Fanuc KAREL source: ko00137.KL

-- PROVISIONAL review KL for V940-1; original PC SHA256 c9733091d5a9caca642406f4a9e78df2e7f2884af441e8ad751a3b0832e9d3ab
-- Incomplete behavior may be omitted. Consult companion uncertainty JSON. Do not deploy.
PROGRAM KO00137
%NOLOCKGROUP
VAR
  R : REAL
  N : INTEGER
-- UNRESOLVED_DECL CFG type=00001c
-- UNRESOLVED_DECL OUT type=000102
BEGIN
  -- V9_ZERO_TABLE_METADATA_HINT layout=0001; no indexed target words; source/name/runtime held
  -- UNRESOLVED_PC offsets 5-12; opcodes 9D,23
  -- UNRESOLVED_PC offsets 17-28; opcodes 2E,23
  -- UNRESOLVED_PC offsets 33-43; opcodes 9D,22,A5
  -- UNRESOLVED_PC offsets 48-107; opcodes 27,22,22,27,21,64,22,22,22,22,76,7E,4A
  -- UNRESOLVED_PC offsets 112-116; opcodes 7F
END KO00137
